Universal Robots PolyScope program: kg_client.urp

Program kg_client (installation=default directory=/programs/usbdisk createdIn=3.3.4.310 lastSavedIn=3.8.0.61336 robotSerialNumber=2018350727)
Calibrated DH parameters: a=[0.000042, -0.345508, -0.391197, 0.000142, -0.000025, 0]; d=[0.089456, 755.785753, -749.950133, -5.725355, 0.095036, 0.082501]; alpha=[1.570684, -0.000328, 0.005444, 1.570522, -1.570384, 0]; deltaTheta=[0.000032, -0.622005, 0.703068, -0.081002, -0.000006, 0.000076]
BeforeStart
  var_1 := False
  thread_flag := False
  var_10 := [0,0,0,0,0,0,0,0,0,0]
  Set NoAction tcp=TCP
Robot Program (runOnlyOnce=false)
  Loop While (checkContinuously=false) expression=var_1==False
    var_1 := socket_open("192.168.1.5",30020)
    Wait Sleep waitTime=0.5
  Loop While (checkContinuously=true) expression=var_1== True
    Wait Sleep waitTime=0.001
    var_2 := socket_read_ascii_float(12)
    Loop While (checkContinuously=false) expression=var_2[0]≠12
      var_2 := socket_read_ascii_float(12)
    Switch expression=var_2[1]
      Case (caseValue=0)
        'movejl'
        var_3 := p[var_2[2],var_2[3],var_2[4],var_2[5],var_2[6],var_2[7]]
        Script: movej(var_3,var_2[8],var_2[9],var_2[10],var_2[11])
        If var_2[12]==0
          Script: socket_send_string("completed_pose_move")
      Case (caseValue=1)
        'movej'
        var_6 := [var_2[2],var_2[3],var_2[4],var_2[5],var_2[6],var_2[7]]
        Script: movej(var_6,var_2[8],var_2[9],var_2[10],var_2[11])
        If var_2[12]==0
          Script: socket_send_string("completed_joint_move")
      Case (caseValue=2)
        'movel'
        var_3 := p[var_2[2],var_2[3],var_2[4],var_2[5],var_2[6],var_2[7]]
        Script: movel(var_3,var_2[8],var_2[9],var_2[10],var_2[11])
        If var_2[12]==0
          Script: socket_send_string("completed_linear_move")
      Case (caseValue=3)
        'move to var_3 relative to current pose'
        var_3 := p[var_2[2],var_2[3],var_2[4],var_2[5],var_2[6],var_2[7]]
        var_5 := get_actual_tcp_pose()
        Script: movel(pose_trans(var_5,var_3),var_2[8],var_2[9],var_2[10],var_2[11])
        If var_2[12]==0
          Script: socket_send_string("completed_relative_linear_move")
      Case (caseValue=4)
        'force move in single axis'
        var_5 := get_actual_tcp_pose()
        If var_2[2]≠0
          Script: var_5[0]=var_5[0]+var_2[2]
          axis := 0
        ElseIf var_2[3]≠0
          Script: var_5[1]=var_5[1]+var_2[3]
          axis := 1
        ElseIf var_2[4]≠0
          Script: var_5[2]=var_5[2]+var_2[4]
          axis := 2
        Script: thread_flag= True
        Loop While (checkContinuously=true) expression=thread_flag== True
          Script: movel(var_5,var_2[8],var_2[9],0,0)
          Wait Sleep waitTime=0.01
          Script: thread_flag= False
        Script: stopl(10)
        If var_2[12]==0
          Script: socket_send_string("completed_force_move")
      Case (caseValue=5)
        'movel'
        var_3 := p[var_2[2],var_2[3],var_2[4],var_2[5],var_2[6],var_2[7]]
        If var_2[12]==0
          Script: stopl(0.5)
        Else 
          Script: movep(var_3,var_2[8],var_2[9],var_2[11])
        If var_2[12]==0
          Script: socket_send_string("completed_linear_move")
      Case (caseValue=10)
        'return current pose'
        var_5 := get_actual_tcp_pose()
        Script: socket_send_string(var_5)
      Case (caseValue=11)
        'return current joints'
        var_4 := get_actual_joint_positions()
        Script: socket_send_string(var_4)
      Case (caseValue=12)
        'return inverse kin of pose'
        var_3 := p[var_2[2],var_2[3],var_2[4],var_2[5],var_2[6],var_2[7]]
        Script: socket_send_string(get_inverse_kin(var_3))
      Case (caseValue=13)
        'return translation to get to 2nd pose from 1st pose coord system'
        var_3 := p[var_2[2],var_2[3],var_2[4],var_2[5],var_2[6],var_2[7]]
        var_5 := get_actual_tcp_pose()
        Script: socket_send_string(pose_trans(var_5,var_3))
      Case (caseValue=14)
        'return current forces'
        Script: socket_send_string(get_tcp_force())
      Case (caseValue=15)
        'return force magnitude'
        Script: socket_send_string(force())
      Case (caseValue=20)
        'set tcp'
        var_3 := p[var_2[2],var_2[3],var_2[4],var_2[5],var_2[6],var_2[7]]
        Script: set_tcp(var_3)
        If var_2[12]==0
          Script: socket_send_string("tcp_updated")
      Case (caseValue=21)
        'set payload'
        Script: set_payload(var_2[8],[var_2[2],var_2[3],var_2[4]])
        If var_2[12]==0
          Script: socket_send_string("payload_updated")
      Case (caseValue=30)
        Script: freedrive_mode()
        Script: socket_send_string("begin_freedrive_mode")
      Case (caseValue=31)
        Script: end_freedrive_mode()
        Script: socket_send_string("end_freedrive_mode")
      Case (caseValue=32)
        Script: socket_send_string("begin_blend_move")
        var_13 := var_2[8]
        n := 0
        Loop While (checkContinuously=false) expression=n<var_13
          Script: n=n+1
          Loop While (checkContinuously=false) expression=var_2[0]≠12
            var_2 := socket_read_ascii_float(12)
          var_3 := p[var_2[2],var_2[3],var_2[4],var_2[5],var_2[6],var_2[7]]
          Script: var_10[n] = var_3
        Script: movel(var_10[0],0.1,0.5,0,0)
        n := 0
        Loop While (checkContinuously=false) expression=n<var_13
          Script: n=n+1
          Script: movep(var_10[n])
      Case (caseValue=33)
        Script: socket_send_string("begin_blend_move")
      Case (caseValue=100)
        'reset program'
        If var_2[12]==0
          Script: socket_send_string("resetting...")
        Script: socket_close()
        var_1 := False
      Case (caseValue=101)
        Script: socket_send_string("ready")
      Case (caseValue=400)
        'safe move'
        var_3 := p[var_2[2],var_2[3],var_2[4],var_2[5],var_2[6],var_2[7]]
        var_5 := get_actual_tcp_pose()
        var_7 := get_inverse_kin(var_3)
        var_8 := get_inverse_kin(var_5)
        var_9 := 0
        Loop Counting (count=6) loopVariable(name=Loop_5)
          If (var_7[Loop_5]-var_8[Loop_5])>2.0  or  (var_8[Loop_5]-var_7[Loop_5])>2.0
            Script: var_9=1
            SuppressedNode
              Script: break
        If var_9==0
          Script: movej(var_3,1,var_2[8],0,0)
          Script: socket_send_string("completed_pose_move")
        Else 
          Script: socket_send_string("no_safe_move_found")
    SuppressedNode
      Wait Sleep waitTime=20
Thread Thread_1 (runOnlyOnce=false trackProgramExecution=false)
  Loop While (checkContinuously=false) expression=thread_flag== False
    Script: var_12=0
    Wait Sleep waitTime=0.01
  Wait Sleep waitTime=0.001
  var_11 := get_tcp_force()
  If var_11[axis]*var_11[axis]<var_2[11]*var_2[11]
    Script: var_12=0
  Else 
    Script: var_12=var_12+1
    If var_12>0
      Script: thread_flag= False
      SuppressedNode
        Script: stopl(1)
      SuppressedNode
        Script: speedl([0,0,0,0,0,0],1,0)
